// TIA Portal V20 export
DATA_BLOCK "ControlNodes"   // DB84
// stored: MemoryReserve 100, Namespace Unit1.Em8
   VAR
      em : "LAF_typeEmControlNode";
      emstate { S7_SetPoint := 'True'} : "LUC_typeStates";
      cm : "Unit1.Em8.typeCmControlNode";
      citiMap : Struct
         PMC : "LER_PMC_Input_Data";
         FlexNet { S7_SetPoint := 'True'} : "LER_FlexNet_Data";
      END_STRUCT;
      hipotThickness : "Unit1.Em8.typeSequenceControlNode";
      GRnR_hipotThickness { S7_SetPoint := 'True'} : "Unit1.Em8.typeSequenceControlNode_GRnR";
      emData : "LER_typePartData";
      SpecialFunctionMode : Struct
         DryRun : Struct
            JRdetectPV : Array[0..15] of Bool;
         END_STRUCT;
      END_STRUCT;
      cmHipotThicknessSafetyPin : "LBC_typeDigitalSignalControlNode";
      cmHipotThicknessJRDetect : "LBC_typeDigitalSignalControlNode";
      cmThicknessAxisZ : "LBC_typeAxis64PosControlNode";
      cmHipotThicknessStageLiftFrontUpDown : "LBC_typeTwoWayActuatorControlNode";
      cmHipotThicknessStageLiftRearUpDown : "LBC_typeTwoWayActuatorControlNode";
      cmHipotTabContactorBwdFwd : "LBC_typeTwoWayActuatorControlNode";
      cmHipotTabContactorLeftOpenClose : "LBC_typeTwoWayActuatorControlNode";
      cmHipotTabContactorRightOpenClose : "LBC_typeTwoWayActuatorControlNode";
      cmHipotThicknessStageLiftAllUpDown : "LBC_typeTwoWayActuatorControlNode";
      cmHipotThicknessServoPress : "LER_typeServoPressControlNode";
      cmThicknessControl : "LER_typeThicknessControlNode";
      cmHipotControl : "LER_typeHipotControlNodes";
   END_VAR
BEGIN
END_DATA_BLOCK
